// TIA Portal V17 export
// export: Created 2024-09-15T12:29:58.742967Z, ExportSetting WithDefaults, DisplayName Totally Integrated Automation Portal, DisplayVersion V17, DisplayName TIA Portal Openness, DisplayVersion V17, DisplayName TIA Portal Version Control Interface, DisplayVersion V17, DisplayName STEP 7 Professional, DisplayVersion V17, DisplayName STEP 7 Safety, DisplayVersion V17, DisplayName WinCC Professional, DisplayVersion V17
DATA_BLOCK "gtyp_SetupAxis"   // DB4
TITLE = Global DB Setup Axis
{ S7_Optimized_Access := 'TRUE' }
AUTHOR : A.Schaefer
VERSION : 0.0
// stored: AutoNumber true, DBAccessibleFromOPCUA true, DBAccessibleFromWebserver true, InstanceOfName typ_SetupAxis, InstanceOfType UDT, IsOnlyStoredInLoadMemory false, IsWriteProtectedInAS false
"typ_SetupAxis"
   // VAR
   //    x_Setup_Activ : Bool;
   //    i_AxisSelection : Int;
   //    i_Function : Int;
   //    x_Set_Ref_Pos : Bool;
   //    x_Set_Soft_End_Pos : Bool;
   //    x_Approach_Ref_Pos : Bool;
   //    x_Axis_Pos : Bool;
   //    x_Axis_Neg : Bool;
   //    x_Approach_Target_Pos : Bool;
   //    w_Increment : Word;
   //    i_PWM : Int;
   //    di_Target_Position : DInt;
   //    di_ActualPosition : DInt;
   //    di_Ref_Pos : DInt;
   //    di_Actual_Ref_Pos : DInt;
   //    di_Soft_End_Pos_Neg : DInt;
   //    di_Actual_Soft_End_Pos_Neg : DInt;
   //    di_Soft_End_Pos_Pos : DInt;
   //    di_Actual_Soft_End_Pos_Pos : DInt;
   //    di_LoopValue : DInt;
   // END_VAR
BEGIN
END_DATA_BLOCK
